// TIA Portal V17 export
// export: Created 2025-03-13T10:29:32.2184254Z, ExportSetting WithDefaults, DisplayName Totally Integrated Automation Portal, DisplayVersion V17 Update 8, DisplayName TIA Portal Openness, DisplayVersion V17 Update 8, DisplayName TIA Portal Version Control Interface, DisplayVersion V17, DisplayName SINAMICS Startdrive Advanced, DisplayVersion V17 SP2, DisplayName SINAMICS Startdrive G110M, G120, G120C, G120D, G120P, G115D, DisplayVersion V17 SP2, DisplayName SINAMICS Startdrive G130, G150, S120, S150, SINAMICS MV, S210, DisplayVersion V17 SP2, DisplayName STEP 7 Professional, DisplayVersion V17 Update 8, DisplayName SINUMERIK ONE STEP 7 Toolbox, DisplayVersion V17 Update 12, DisplayName SINUMERIK 840D sl STEP 7 Toolbox, DisplayVersion V17 Update 12, DisplayName STEP 7 Safety, DisplayVersion V17 Update 6, DisplayName WinCC Advanced, DisplayVersion V17 Update 8
FUNCTION_BLOCK "FB1801_STA3_CLEANING_VALVE"   // FB1801, LAD
{ S7_Optimized_Access := 'TRUE' }
VERSION : 0.1
// stored: AutoNumber false, IsIECCheckEnabled false, IsRetainMemResEnabled false, MemoryReserve 100, SetENOAutomatically false, UDAEnableTagReadback false
   VAR_INPUT
      SWITCH_ON_GEN_CON : Bool;
      SWITCH_ON_CON : Bool;
      SWITCH_ON_AUTO_REQ : Bool;
      SWITCH_OFF_CON : Bool;
      SWITCH_OFF_AUTO_REQ : Bool;
      HMI_LINE_REQ : Bool;
      UNIT_ALARM : UInt;
      STATION_ALARM : UInt;
   END_VAR
   VAR_OUTPUT
      SWITCHED_ON : Bool;
      SWITCHED_OFF : Bool;
      HMI_MOTION_EXECUTABILITY_LEFT : Bool;
      HMI_MOTION_EXECUTABILITY_RIGHT : Bool;
      HMI_MOTION_END_POS_LEFT : Bool;
      HMI_MOTION_END_POS_RIGHT : Bool;
      SWITCH_ON : Bool;
      SWITCH_OFF : Bool;
   END_VAR
   VAR
      VALVE : "ASPIRATION";
   END_VAR
   VAR DB_SPECIFIC
      TIMER_SIMULTANEITY { S7_SetPoint := 'True'} : TON_TIME;   // SIMULTANEITY TIMER
      TIMER_TIME_EXCEEDED { S7_SetPoint := 'True'} : TON_TIME;   // TIME EXCEEDED TIMER
   END_VAR
   VAR_TEMP
      DB_NUMBER : DInt;   // DB NUMBER FOR ALARM AND HELP DECODING
   END_VAR
   // TIMER_SIMULTANEITY.PT := T#100MS;
   // TIMER_TIME_EXCEEDED.PT := T#8S;
   VAR_TEMP   // added for the SCL form of the ladder/FBD networks
      _w1 : Bool;
      _w2 : Bool;
   END_VAR
BEGIN

REGION Network 1: GENERAL CONDITIONS
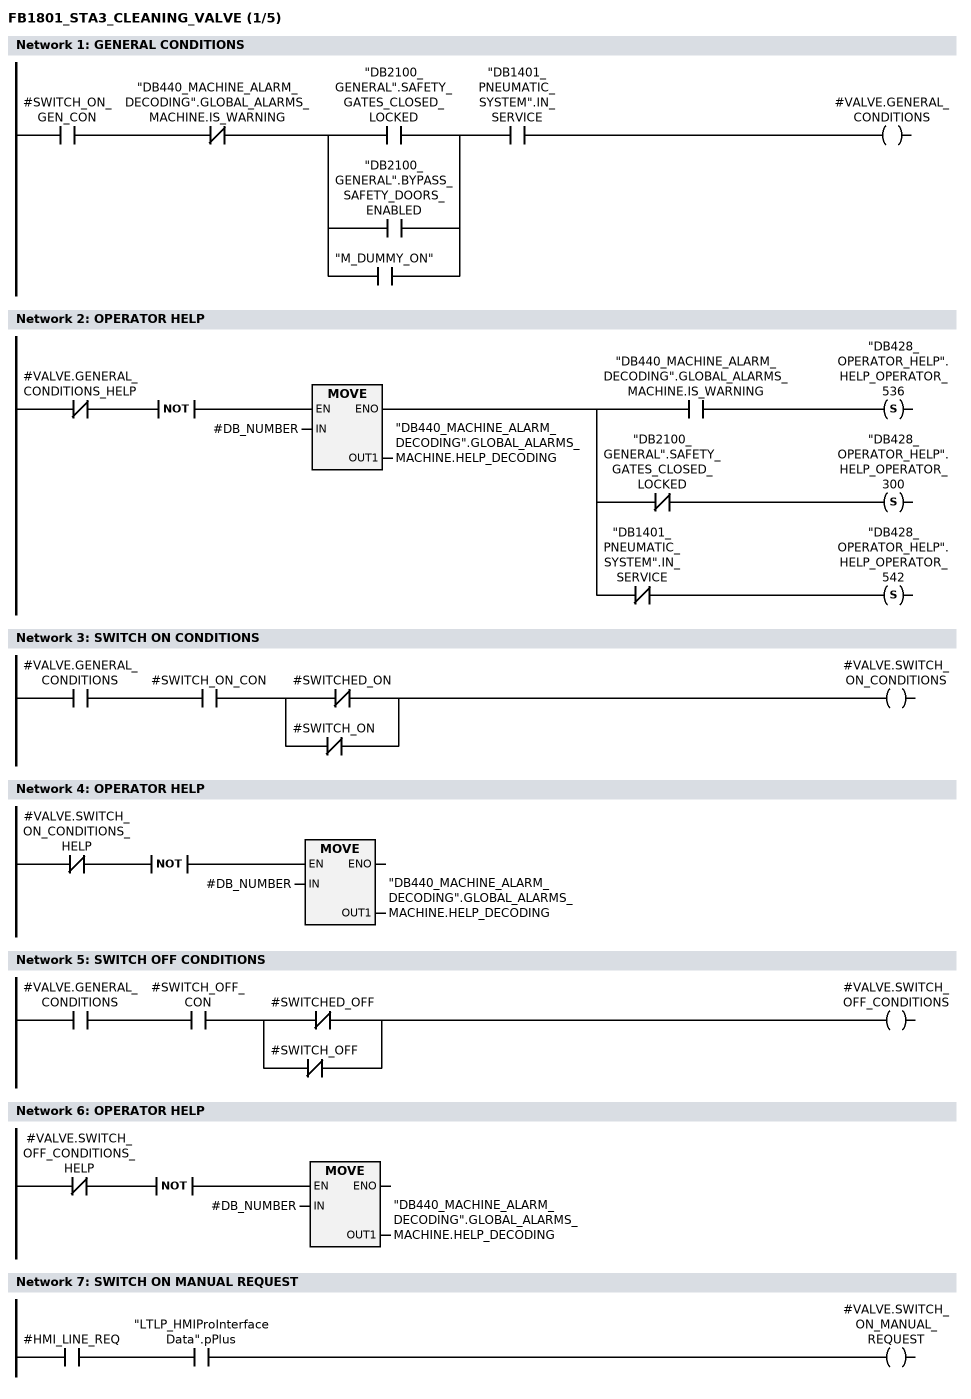
   RUNG wire#powerrail
      Contact( #SWITCH_ON_GEN_CON )
      I_Contact( "DB440_MACHINE_ALARM_DECODING".GLOBAL_ALARMS_MACHINE.IS_WARNING )
      wire#w1
      Contact( "DB2100_GENERAL".SAFETY_GATES_CLOSED_LOCKED )
      wire#w2
      Contact( "DB1401_PNEUMATIC_SYSTEM".IN_SERVICE )
      Coil( #VALVE.GENERAL_CONDITIONS )
   END_RUNG
   RUNG wire#w1
      Contact( "DB2100_GENERAL".BYPASS_SAFETY_DOORS_ENABLED )
   END_RUNG wire#w2
   RUNG wire#w1
      Contact( "M_DUMMY_ON" )
   END_RUNG wire#w2
   // the same network as SCL:
   #VALVE.GENERAL_CONDITIONS := #SWITCH_ON_GEN_CON AND NOT "DB440_MACHINE_ALARM_DECODING".GLOBAL_ALARMS_MACHINE.IS_WARNING AND ("DB2100_GENERAL".SAFETY_GATES_CLOSED_LOCKED OR "DB2100_GENERAL".BYPASS_SAFETY_DOORS_ENABLED OR "M_DUMMY_ON") AND "DB1401_PNEUMATIC_SYSTEM".IN_SERVICE;
END_REGION

REGION Network 2: OPERATOR HELP
   RUNG wire#powerrail
      I_Contact( #VALVE.GENERAL_CONDITIONS_HELP )
      Not()
      { S7_GenerateENO := "TRUE" } Move(in := #DB_NUMBER, out1 => "DB440_MACHINE_ALARM_DECODING".GLOBAL_ALARMS_MACHINE.HELP_DECODING)
      wire#w1
      Contact( "DB440_MACHINE_ALARM_DECODING".GLOBAL_ALARMS_MACHINE.IS_WARNING )
      S_Coil( "DB428_OPERATOR_HELP".HELP_OPERATOR_536 )
   END_RUNG
   RUNG wire#w1
      I_Contact( "DB2100_GENERAL".SAFETY_GATES_CLOSED_LOCKED )
      S_Coil( "DB428_OPERATOR_HELP".HELP_OPERATOR_300 )
   END_RUNG
   RUNG wire#w1
      I_Contact( "DB1401_PNEUMATIC_SYSTEM".IN_SERVICE )
      S_Coil( "DB428_OPERATOR_HELP".HELP_OPERATOR_542 )
   END_RUNG
   // the same network as SCL:
   // ENO of a box is taken as its EN; it also drops when the box reports an error
   #_w1 := NOT (NOT #VALVE.GENERAL_CONDITIONS_HELP);
   IF #_w1 THEN "DB440_MACHINE_ALARM_DECODING".GLOBAL_ALARMS_MACHINE.HELP_DECODING := #DB_NUMBER; END_IF;
   IF #_w1 AND "DB440_MACHINE_ALARM_DECODING".GLOBAL_ALARMS_MACHINE.IS_WARNING THEN
       "DB428_OPERATOR_HELP".HELP_OPERATOR_536 := TRUE;
   END_IF;
   IF #_w1 AND NOT "DB2100_GENERAL".SAFETY_GATES_CLOSED_LOCKED THEN
       "DB428_OPERATOR_HELP".HELP_OPERATOR_300 := TRUE;
   END_IF;
   IF #_w1 AND NOT "DB1401_PNEUMATIC_SYSTEM".IN_SERVICE THEN
       "DB428_OPERATOR_HELP".HELP_OPERATOR_542 := TRUE;
   END_IF;
END_REGION

REGION Network 3: SWITCH ON CONDITIONS
   RUNG wire#powerrail
      Contact( #VALVE.GENERAL_CONDITIONS )
      Contact( #SWITCH_ON_CON )
      wire#w1
      I_Contact( #SWITCHED_ON )
      wire#w2
      Coil( #VALVE.SWITCH_ON_CONDITIONS )
   END_RUNG
   RUNG wire#w1
      I_Contact( #SWITCH_ON )
   END_RUNG wire#w2
   // the same network as SCL:
   #VALVE.SWITCH_ON_CONDITIONS := #VALVE.GENERAL_CONDITIONS AND #SWITCH_ON_CON AND (NOT #SWITCHED_ON OR NOT #SWITCH_ON);
END_REGION

REGION Network 4: OPERATOR HELP
   RUNG wire#powerrail
      I_Contact( #VALVE.SWITCH_ON_CONDITIONS_HELP )
      Not()
      { S7_GenerateENO := "TRUE" } Move(in := #DB_NUMBER, out1 => "DB440_MACHINE_ALARM_DECODING".GLOBAL_ALARMS_MACHINE.HELP_DECODING)
   END_RUNG
   // the same network as SCL:
   IF NOT (NOT #VALVE.SWITCH_ON_CONDITIONS_HELP) THEN
       "DB440_MACHINE_ALARM_DECODING".GLOBAL_ALARMS_MACHINE.HELP_DECODING := #DB_NUMBER;
   END_IF;
END_REGION

REGION Network 5: SWITCH OFF CONDITIONS
   RUNG wire#powerrail
      Contact( #VALVE.GENERAL_CONDITIONS )
      Contact( #SWITCH_OFF_CON )
      wire#w1
      I_Contact( #SWITCHED_OFF )
      wire#w2
      Coil( #VALVE.SWITCH_OFF_CONDITIONS )
   END_RUNG
   RUNG wire#w1
      I_Contact( #SWITCH_OFF )
   END_RUNG wire#w2
   // the same network as SCL:
   #VALVE.SWITCH_OFF_CONDITIONS := #VALVE.GENERAL_CONDITIONS AND #SWITCH_OFF_CON AND (NOT #SWITCHED_OFF OR NOT #SWITCH_OFF);
END_REGION

REGION Network 6: OPERATOR HELP
   RUNG wire#powerrail
      I_Contact( #VALVE.SWITCH_OFF_CONDITIONS_HELP )
      Not()
      { S7_GenerateENO := "TRUE" } Move(in := #DB_NUMBER, out1 => "DB440_MACHINE_ALARM_DECODING".GLOBAL_ALARMS_MACHINE.HELP_DECODING)
   END_RUNG
   // the same network as SCL:
   IF NOT (NOT #VALVE.SWITCH_OFF_CONDITIONS_HELP) THEN
       "DB440_MACHINE_ALARM_DECODING".GLOBAL_ALARMS_MACHINE.HELP_DECODING := #DB_NUMBER;
   END_IF;
END_REGION

REGION Network 7: SWITCH ON MANUAL REQUEST
   RUNG wire#powerrail
      Contact( #HMI_LINE_REQ )
      Contact( "LTLP_HMIProInterfaceData".pPlus )
      Coil( #VALVE.SWITCH_ON_MANUAL_REQUEST )
   END_RUNG
   // the same network as SCL:
   #VALVE.SWITCH_ON_MANUAL_REQUEST := #HMI_LINE_REQ AND "LTLP_HMIProInterfaceData".pPlus;
END_REGION

REGION Network 8: SWITCH OFF MANUAL REQUEST
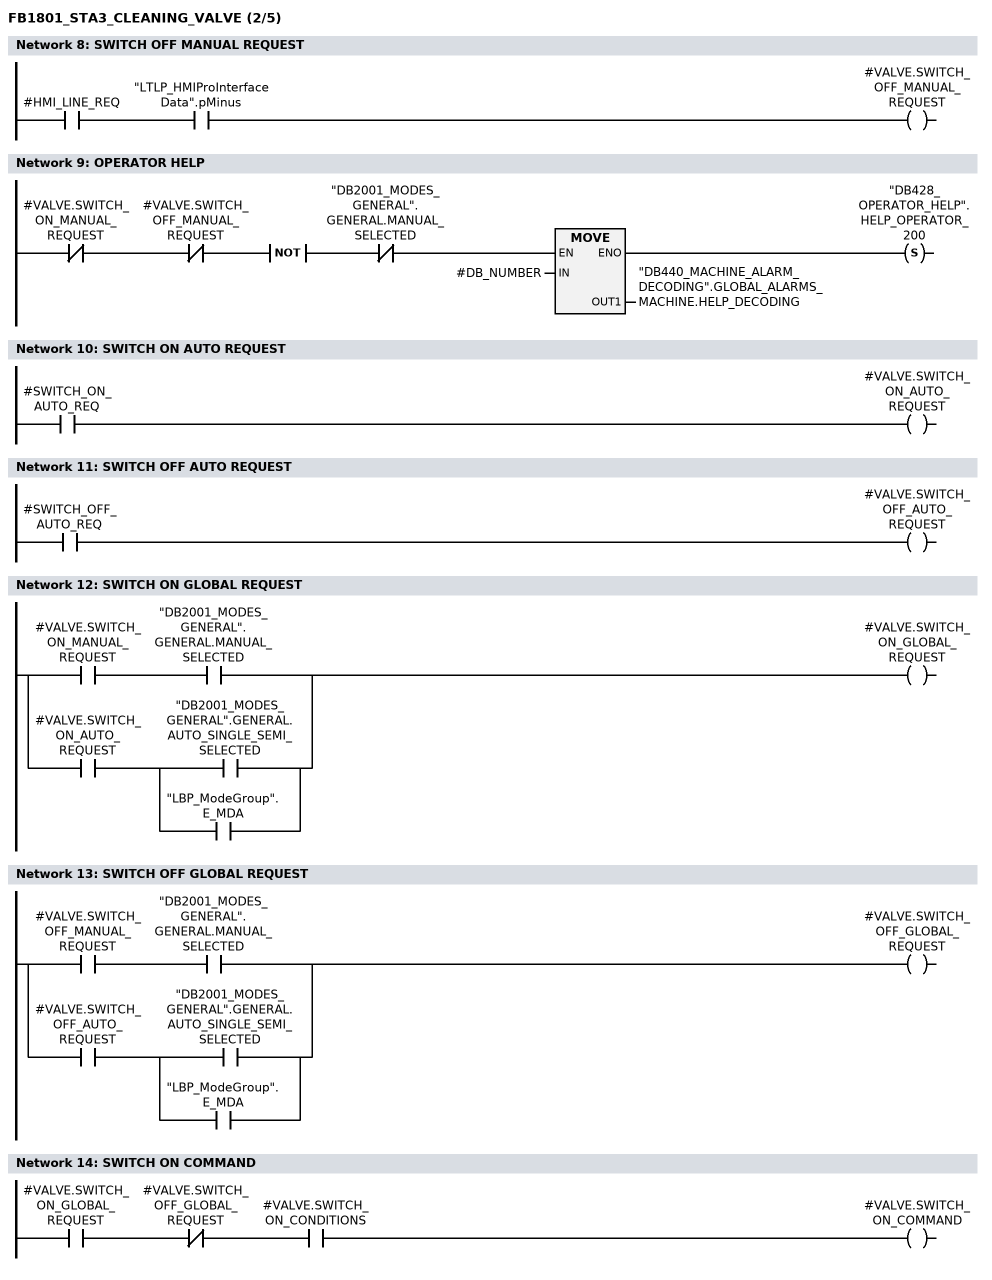
   RUNG wire#powerrail
      Contact( #HMI_LINE_REQ )
      Contact( "LTLP_HMIProInterfaceData".pMinus )
      Coil( #VALVE.SWITCH_OFF_MANUAL_REQUEST )
   END_RUNG
   // the same network as SCL:
   #VALVE.SWITCH_OFF_MANUAL_REQUEST := #HMI_LINE_REQ AND "LTLP_HMIProInterfaceData".pMinus;
END_REGION

REGION Network 9: OPERATOR HELP
   RUNG wire#powerrail
      I_Contact( #VALVE.SWITCH_ON_MANUAL_REQUEST )
      I_Contact( #VALVE.SWITCH_OFF_MANUAL_REQUEST )
      Not()
      I_Contact( "DB2001_MODES_GENERAL".GENERAL.MANUAL_SELECTED )
      { S7_GenerateENO := "TRUE" } Move(in := #DB_NUMBER, out1 => "DB440_MACHINE_ALARM_DECODING".GLOBAL_ALARMS_MACHINE.HELP_DECODING)
      S_Coil( "DB428_OPERATOR_HELP".HELP_OPERATOR_200 )
   END_RUNG
   // the same network as SCL:
   // ENO of a box is taken as its EN; it also drops when the box reports an error
   IF NOT (NOT #VALVE.SWITCH_ON_MANUAL_REQUEST AND NOT #VALVE.SWITCH_OFF_MANUAL_REQUEST) AND NOT "DB2001_MODES_GENERAL".GENERAL.MANUAL_SELECTED THEN
       "DB440_MACHINE_ALARM_DECODING".GLOBAL_ALARMS_MACHINE.HELP_DECODING := #DB_NUMBER;
       "DB428_OPERATOR_HELP".HELP_OPERATOR_200 := TRUE;
   END_IF;
END_REGION

REGION Network 10: SWITCH ON AUTO REQUEST
   RUNG wire#powerrail
      Contact( #SWITCH_ON_AUTO_REQ )
      Coil( #VALVE.SWITCH_ON_AUTO_REQUEST )
   END_RUNG
   // the same network as SCL:
   #VALVE.SWITCH_ON_AUTO_REQUEST := #SWITCH_ON_AUTO_REQ;
END_REGION

REGION Network 11: SWITCH OFF AUTO REQUEST
   RUNG wire#powerrail
      Contact( #SWITCH_OFF_AUTO_REQ )
      Coil( #VALVE.SWITCH_OFF_AUTO_REQUEST )
   END_RUNG
   // the same network as SCL:
   #VALVE.SWITCH_OFF_AUTO_REQUEST := #SWITCH_OFF_AUTO_REQ;
END_REGION

REGION Network 12: SWITCH ON GLOBAL REQUEST
   RUNG wire#powerrail
      Contact( #VALVE.SWITCH_ON_MANUAL_REQUEST )
      Contact( "DB2001_MODES_GENERAL".GENERAL.MANUAL_SELECTED )
      wire#w1
      Coil( #VALVE.SWITCH_ON_GLOBAL_REQUEST )
   END_RUNG
   RUNG wire#powerrail
      Contact( #VALVE.SWITCH_ON_AUTO_REQUEST )
      wire#w2
      Contact( "DB2001_MODES_GENERAL".GENERAL.AUTO_SINGLE_SEMI_SELECTED )
   END_RUNG wire#w1
   RUNG wire#w2
      Contact( "LBP_ModeGroup".E_MDA )
   END_RUNG wire#w1
   // the same network as SCL:
   #VALVE.SWITCH_ON_GLOBAL_REQUEST := (#VALVE.SWITCH_ON_MANUAL_REQUEST AND "DB2001_MODES_GENERAL".GENERAL.MANUAL_SELECTED) OR (#VALVE.SWITCH_ON_AUTO_REQUEST AND ("DB2001_MODES_GENERAL".GENERAL.AUTO_SINGLE_SEMI_SELECTED OR "LBP_ModeGroup".E_MDA));
END_REGION

REGION Network 13: SWITCH OFF GLOBAL REQUEST
   RUNG wire#powerrail
      Contact( #VALVE.SWITCH_OFF_MANUAL_REQUEST )
      Contact( "DB2001_MODES_GENERAL".GENERAL.MANUAL_SELECTED )
      wire#w1
      Coil( #VALVE.SWITCH_OFF_GLOBAL_REQUEST )
   END_RUNG
   RUNG wire#powerrail
      Contact( #VALVE.SWITCH_OFF_AUTO_REQUEST )
      wire#w2
      Contact( "DB2001_MODES_GENERAL".GENERAL.AUTO_SINGLE_SEMI_SELECTED )
   END_RUNG wire#w1
   RUNG wire#w2
      Contact( "LBP_ModeGroup".E_MDA )
   END_RUNG wire#w1
   // the same network as SCL:
   #VALVE.SWITCH_OFF_GLOBAL_REQUEST := (#VALVE.SWITCH_OFF_MANUAL_REQUEST AND "DB2001_MODES_GENERAL".GENERAL.MANUAL_SELECTED) OR (#VALVE.SWITCH_OFF_AUTO_REQUEST AND ("DB2001_MODES_GENERAL".GENERAL.AUTO_SINGLE_SEMI_SELECTED OR "LBP_ModeGroup".E_MDA));
END_REGION

REGION Network 14: SWITCH ON COMMAND
   RUNG wire#powerrail
      Contact( #VALVE.SWITCH_ON_GLOBAL_REQUEST )
      I_Contact( #VALVE.SWITCH_OFF_GLOBAL_REQUEST )
      Contact( #VALVE.SWITCH_ON_CONDITIONS )
      Coil( #VALVE.SWITCH_ON_COMMAND )
   END_RUNG
   // the same network as SCL:
   #VALVE.SWITCH_ON_COMMAND := #VALVE.SWITCH_ON_GLOBAL_REQUEST AND NOT #VALVE.SWITCH_OFF_GLOBAL_REQUEST AND #VALVE.SWITCH_ON_CONDITIONS;
END_REGION

REGION Network 15: SWITCH OFF COMMAND
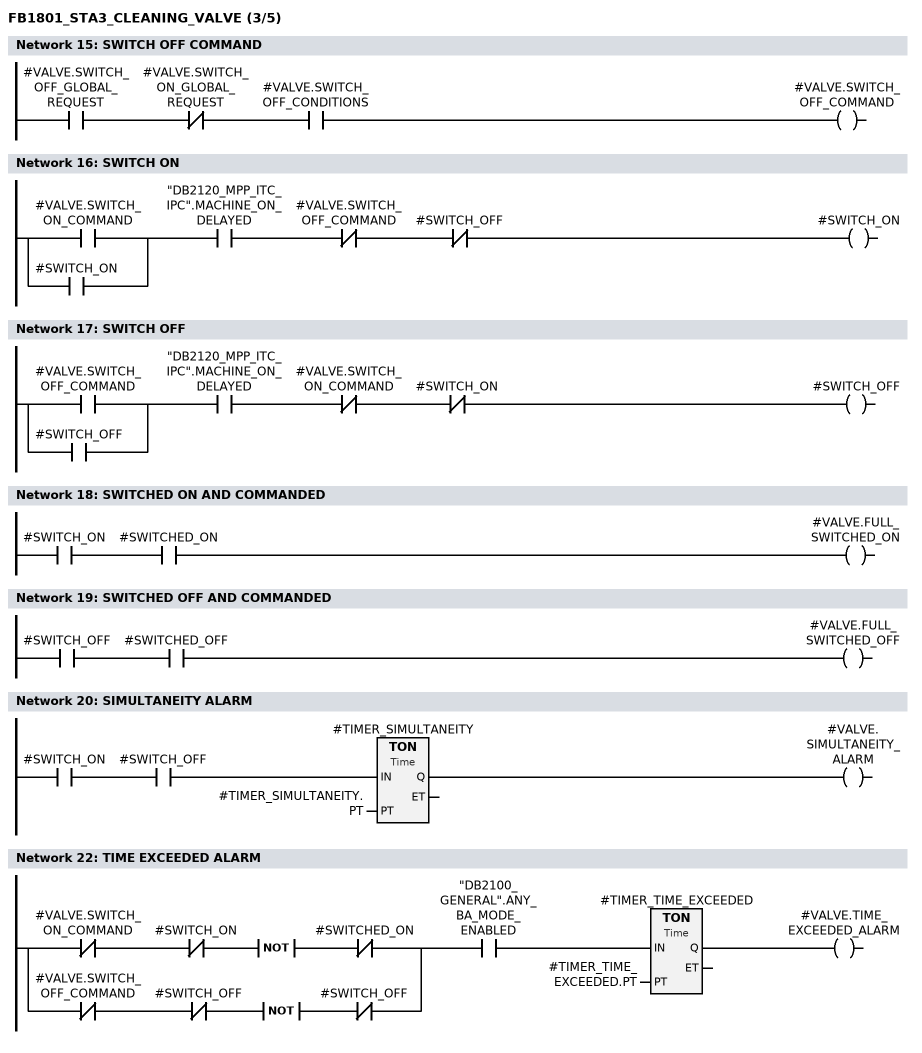
   RUNG wire#powerrail
      Contact( #VALVE.SWITCH_OFF_GLOBAL_REQUEST )
      I_Contact( #VALVE.SWITCH_ON_GLOBAL_REQUEST )
      Contact( #VALVE.SWITCH_OFF_CONDITIONS )
      Coil( #VALVE.SWITCH_OFF_COMMAND )
   END_RUNG
   // the same network as SCL:
   #VALVE.SWITCH_OFF_COMMAND := #VALVE.SWITCH_OFF_GLOBAL_REQUEST AND NOT #VALVE.SWITCH_ON_GLOBAL_REQUEST AND #VALVE.SWITCH_OFF_CONDITIONS;
END_REGION

REGION Network 16: SWITCH ON
   RUNG wire#powerrail
      Contact( #VALVE.SWITCH_ON_COMMAND )
      wire#w1
      Contact( "DB2120_MPP_ITC_IPC".MACHINE_ON_DELAYED )
      I_Contact( #VALVE.SWITCH_OFF_COMMAND )
      I_Contact( #SWITCH_OFF )
      Coil( #SWITCH_ON )
   END_RUNG
   RUNG wire#powerrail
      Contact( #SWITCH_ON )
   END_RUNG wire#w1
   // the same network as SCL:
   #SWITCH_ON := (#VALVE.SWITCH_ON_COMMAND OR #SWITCH_ON) AND "DB2120_MPP_ITC_IPC".MACHINE_ON_DELAYED AND NOT #VALVE.SWITCH_OFF_COMMAND AND NOT #SWITCH_OFF;
END_REGION

REGION Network 17: SWITCH OFF
   RUNG wire#powerrail
      Contact( #VALVE.SWITCH_OFF_COMMAND )
      wire#w1
      Contact( "DB2120_MPP_ITC_IPC".MACHINE_ON_DELAYED )
      I_Contact( #VALVE.SWITCH_ON_COMMAND )
      I_Contact( #SWITCH_ON )
      Coil( #SWITCH_OFF )
   END_RUNG
   RUNG wire#powerrail
      Contact( #SWITCH_OFF )
   END_RUNG wire#w1
   // the same network as SCL:
   #SWITCH_OFF := (#VALVE.SWITCH_OFF_COMMAND OR #SWITCH_OFF) AND "DB2120_MPP_ITC_IPC".MACHINE_ON_DELAYED AND NOT #VALVE.SWITCH_ON_COMMAND AND NOT #SWITCH_ON;
END_REGION

REGION Network 18: SWITCHED ON AND COMMANDED
   RUNG wire#powerrail
      Contact( #SWITCH_ON )
      Contact( #SWITCHED_ON )
      Coil( #VALVE.FULL_SWITCHED_ON )
   END_RUNG
   // the same network as SCL:
   #VALVE.FULL_SWITCHED_ON := #SWITCH_ON AND #SWITCHED_ON;
END_REGION

REGION Network 19: SWITCHED OFF AND COMMANDED
   RUNG wire#powerrail
      Contact( #SWITCH_OFF )
      Contact( #SWITCHED_OFF )
      Coil( #VALVE.FULL_SWITCHED_OFF )
   END_RUNG
   // the same network as SCL:
   #VALVE.FULL_SWITCHED_OFF := #SWITCH_OFF AND #SWITCHED_OFF;
END_REGION

REGION Network 20: SIMULTANEITY ALARM
   RUNG wire#powerrail
      Contact( #SWITCH_ON )
      Contact( #SWITCH_OFF )
      { S7_Templates := "time_type := Time" } #TIMER_SIMULTANEITY.TON(pt := #TIMER_SIMULTANEITY.PT, et =>)
      Coil( #VALVE.SIMULTANEITY_ALARM )
   END_RUNG
   // the same network as SCL:
   #TIMER_SIMULTANEITY(IN := #SWITCH_ON AND #SWITCH_OFF, PT := #TIMER_SIMULTANEITY.PT);   // TON
   #VALVE.SIMULTANEITY_ALARM := #TIMER_SIMULTANEITY.Q;
END_REGION

NETWORK
TITLE = READ INSTANCE DB
      L     DINO;
      +     10#800000;
      T     #DB_NUMBER;


REGION Network 22: TIME EXCEEDED ALARM
   RUNG wire#powerrail
      I_Contact( #VALVE.SWITCH_ON_COMMAND )
      I_Contact( #SWITCH_ON )
      Not()
      I_Contact( #SWITCHED_ON )
      wire#w1
      Contact( "DB2100_GENERAL".ANY_BA_MODE_ENABLED )
      { S7_Templates := "time_type := Time" } #TIMER_TIME_EXCEEDED.TON(pt := #TIMER_TIME_EXCEEDED.PT, et =>)
      Coil( #VALVE.TIME_EXCEEDED_ALARM )
   END_RUNG
   RUNG wire#powerrail
      I_Contact( #VALVE.SWITCH_OFF_COMMAND )
      I_Contact( #SWITCH_OFF )
      Not()
      I_Contact( #SWITCH_OFF )
   END_RUNG wire#w1
   // the same network as SCL:
   #TIMER_TIME_EXCEEDED(IN := ((NOT (NOT #VALVE.SWITCH_ON_COMMAND AND NOT #SWITCH_ON) AND NOT #SWITCHED_ON) OR (NOT (NOT #VALVE.SWITCH_OFF_COMMAND AND NOT #SWITCH_OFF) AND NOT #SWITCH_OFF)) AND "DB2100_GENERAL".ANY_BA_MODE_ENABLED,   // TON
                        PT := #TIMER_TIME_EXCEEDED.PT);
   #VALVE.TIME_EXCEEDED_ALARM := #TIMER_TIME_EXCEEDED.Q;
END_REGION

REGION Network 23: IMMEDIATE STOP AND STOP END OF CYCLE ALARMS
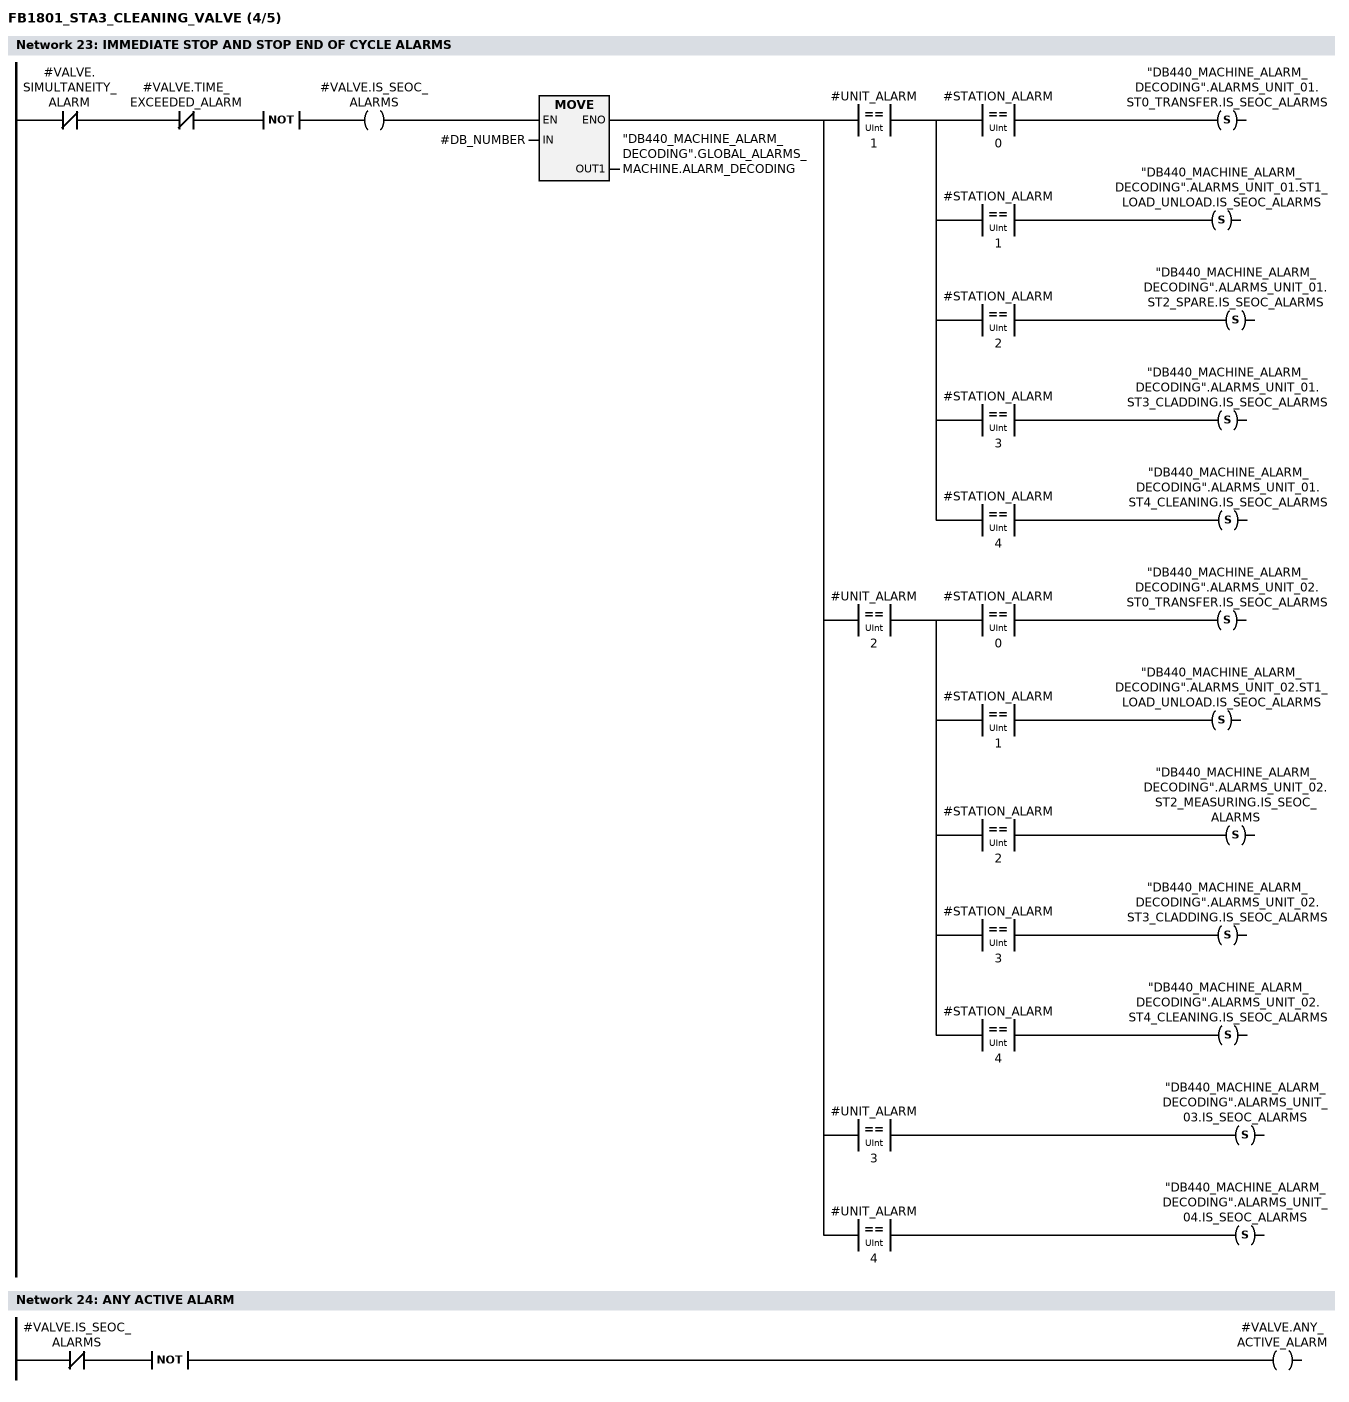
   RUNG wire#powerrail
      I_Contact( #VALVE.SIMULTANEITY_ALARM )
      I_Contact( #VALVE.TIME_EXCEEDED_ALARM )
      Not()
      Coil( #VALVE.IS_SEOC_ALARMS )
      { S7_GenerateENO := "TRUE" } Move(in := #DB_NUMBER, out1 => "DB440_MACHINE_ALARM_DECODING".GLOBAL_ALARMS_MACHINE.ALARM_DECODING)
      wire#w1
      { S7_Templates := "SrcType := UInt" } EQ_Contact(in1 := #UNIT_ALARM, in2 := 1)
      wire#w2
      { S7_Templates := "SrcType := UInt" } EQ_Contact(in1 := #STATION_ALARM, in2 := 0)
      S_Coil( "DB440_MACHINE_ALARM_DECODING".ALARMS_UNIT_01.ST0_TRANSFER.IS_SEOC_ALARMS )
   END_RUNG
   RUNG wire#w2
      { S7_Templates := "SrcType := UInt" } EQ_Contact(in1 := #STATION_ALARM, in2 := 1)
      S_Coil( "DB440_MACHINE_ALARM_DECODING".ALARMS_UNIT_01.ST1_LOAD_UNLOAD.IS_SEOC_ALARMS )
   END_RUNG
   RUNG wire#w2
      { S7_Templates := "SrcType := UInt" } EQ_Contact(in1 := #STATION_ALARM, in2 := 2)
      S_Coil( "DB440_MACHINE_ALARM_DECODING".ALARMS_UNIT_01.ST2_SPARE.IS_SEOC_ALARMS )
   END_RUNG
   RUNG wire#w2
      { S7_Templates := "SrcType := UInt" } EQ_Contact(in1 := #STATION_ALARM, in2 := 3)
      S_Coil( "DB440_MACHINE_ALARM_DECODING".ALARMS_UNIT_01.ST3_CLADDING.IS_SEOC_ALARMS )
   END_RUNG
   RUNG wire#w2
      { S7_Templates := "SrcType := UInt" } EQ_Contact(in1 := #STATION_ALARM, in2 := 4)
      S_Coil( "DB440_MACHINE_ALARM_DECODING".ALARMS_UNIT_01.ST4_CLEANING.IS_SEOC_ALARMS )
   END_RUNG
   RUNG wire#w1
      { S7_Templates := "SrcType := UInt" } EQ_Contact(in1 := #UNIT_ALARM, in2 := 2)
      wire#w3
      { S7_Templates := "SrcType := UInt" } EQ_Contact(in1 := #STATION_ALARM, in2 := 0)
      S_Coil( "DB440_MACHINE_ALARM_DECODING".ALARMS_UNIT_02.ST0_TRANSFER.IS_SEOC_ALARMS )
   END_RUNG
   RUNG wire#w3
      { S7_Templates := "SrcType := UInt" } EQ_Contact(in1 := #STATION_ALARM, in2 := 1)
      S_Coil( "DB440_MACHINE_ALARM_DECODING".ALARMS_UNIT_02.ST1_LOAD_UNLOAD.IS_SEOC_ALARMS )
   END_RUNG
   RUNG wire#w3
      { S7_Templates := "SrcType := UInt" } EQ_Contact(in1 := #STATION_ALARM, in2 := 2)
      S_Coil( "DB440_MACHINE_ALARM_DECODING".ALARMS_UNIT_02.ST2_MEASURING.IS_SEOC_ALARMS )
   END_RUNG
   RUNG wire#w3
      { S7_Templates := "SrcType := UInt" } EQ_Contact(in1 := #STATION_ALARM, in2 := 3)
      S_Coil( "DB440_MACHINE_ALARM_DECODING".ALARMS_UNIT_02.ST3_CLADDING.IS_SEOC_ALARMS )
   END_RUNG
   RUNG wire#w3
      { S7_Templates := "SrcType := UInt" } EQ_Contact(in1 := #STATION_ALARM, in2 := 4)
      S_Coil( "DB440_MACHINE_ALARM_DECODING".ALARMS_UNIT_02.ST4_CLEANING.IS_SEOC_ALARMS )
   END_RUNG
   RUNG wire#w1
      { S7_Templates := "SrcType := UInt" } EQ_Contact(in1 := #UNIT_ALARM, in2 := 3)
      S_Coil( "DB440_MACHINE_ALARM_DECODING".ALARMS_UNIT_03.IS_SEOC_ALARMS )
   END_RUNG
   RUNG wire#w1
      { S7_Templates := "SrcType := UInt" } EQ_Contact(in1 := #UNIT_ALARM, in2 := 4)
      S_Coil( "DB440_MACHINE_ALARM_DECODING".ALARMS_UNIT_04.IS_SEOC_ALARMS )
   END_RUNG
   // the same network as SCL:
   // ENO of a box is taken as its EN; it also drops when the box reports an error
   #VALVE.IS_SEOC_ALARMS := NOT (NOT #VALVE.SIMULTANEITY_ALARM AND NOT #VALVE.TIME_EXCEEDED_ALARM);
   IF #VALVE.IS_SEOC_ALARMS THEN
       "DB440_MACHINE_ALARM_DECODING".GLOBAL_ALARMS_MACHINE.ALARM_DECODING := #DB_NUMBER;
   END_IF;
   #_w1 := #VALVE.IS_SEOC_ALARMS AND (#UNIT_ALARM = 1);
   IF #_w1 AND (#STATION_ALARM = 0) THEN
       "DB440_MACHINE_ALARM_DECODING".ALARMS_UNIT_01.ST0_TRANSFER.IS_SEOC_ALARMS := TRUE;
   END_IF;
   IF #_w1 AND (#STATION_ALARM = 1) THEN
       "DB440_MACHINE_ALARM_DECODING".ALARMS_UNIT_01.ST1_LOAD_UNLOAD.IS_SEOC_ALARMS := TRUE;
   END_IF;
   IF #_w1 AND (#STATION_ALARM = 2) THEN
       "DB440_MACHINE_ALARM_DECODING".ALARMS_UNIT_01.ST2_SPARE.IS_SEOC_ALARMS := TRUE;
   END_IF;
   IF #_w1 AND (#STATION_ALARM = 3) THEN
       "DB440_MACHINE_ALARM_DECODING".ALARMS_UNIT_01.ST3_CLADDING.IS_SEOC_ALARMS := TRUE;
   END_IF;
   IF #_w1 AND (#STATION_ALARM = 4) THEN
       "DB440_MACHINE_ALARM_DECODING".ALARMS_UNIT_01.ST4_CLEANING.IS_SEOC_ALARMS := TRUE;
   END_IF;
   #_w2 := #VALVE.IS_SEOC_ALARMS AND (#UNIT_ALARM = 2);
   IF #_w2 AND (#STATION_ALARM = 0) THEN
       "DB440_MACHINE_ALARM_DECODING".ALARMS_UNIT_02.ST0_TRANSFER.IS_SEOC_ALARMS := TRUE;
   END_IF;
   IF #_w2 AND (#STATION_ALARM = 1) THEN
       "DB440_MACHINE_ALARM_DECODING".ALARMS_UNIT_02.ST1_LOAD_UNLOAD.IS_SEOC_ALARMS := TRUE;
   END_IF;
   IF #_w2 AND (#STATION_ALARM = 2) THEN
       "DB440_MACHINE_ALARM_DECODING".ALARMS_UNIT_02.ST2_MEASURING.IS_SEOC_ALARMS := TRUE;
   END_IF;
   IF #_w2 AND (#STATION_ALARM = 3) THEN
       "DB440_MACHINE_ALARM_DECODING".ALARMS_UNIT_02.ST3_CLADDING.IS_SEOC_ALARMS := TRUE;
   END_IF;
   IF #_w2 AND (#STATION_ALARM = 4) THEN
       "DB440_MACHINE_ALARM_DECODING".ALARMS_UNIT_02.ST4_CLEANING.IS_SEOC_ALARMS := TRUE;
   END_IF;
   IF #VALVE.IS_SEOC_ALARMS AND (#UNIT_ALARM = 3) THEN
       "DB440_MACHINE_ALARM_DECODING".ALARMS_UNIT_03.IS_SEOC_ALARMS := TRUE;
   END_IF;
   IF #VALVE.IS_SEOC_ALARMS AND (#UNIT_ALARM = 4) THEN
       "DB440_MACHINE_ALARM_DECODING".ALARMS_UNIT_04.IS_SEOC_ALARMS := TRUE;
   END_IF;
END_REGION

REGION Network 24: ANY ACTIVE ALARM
   RUNG wire#powerrail
      I_Contact( #VALVE.IS_SEOC_ALARMS )
      Not()
      Coil( #VALVE.ANY_ACTIVE_ALARM )
   END_RUNG
   // the same network as SCL:
   #VALVE.ANY_ACTIVE_ALARM := NOT (NOT #VALVE.IS_SEOC_ALARMS);
END_REGION

REGION Network 25: PROGRAMMING ALARM
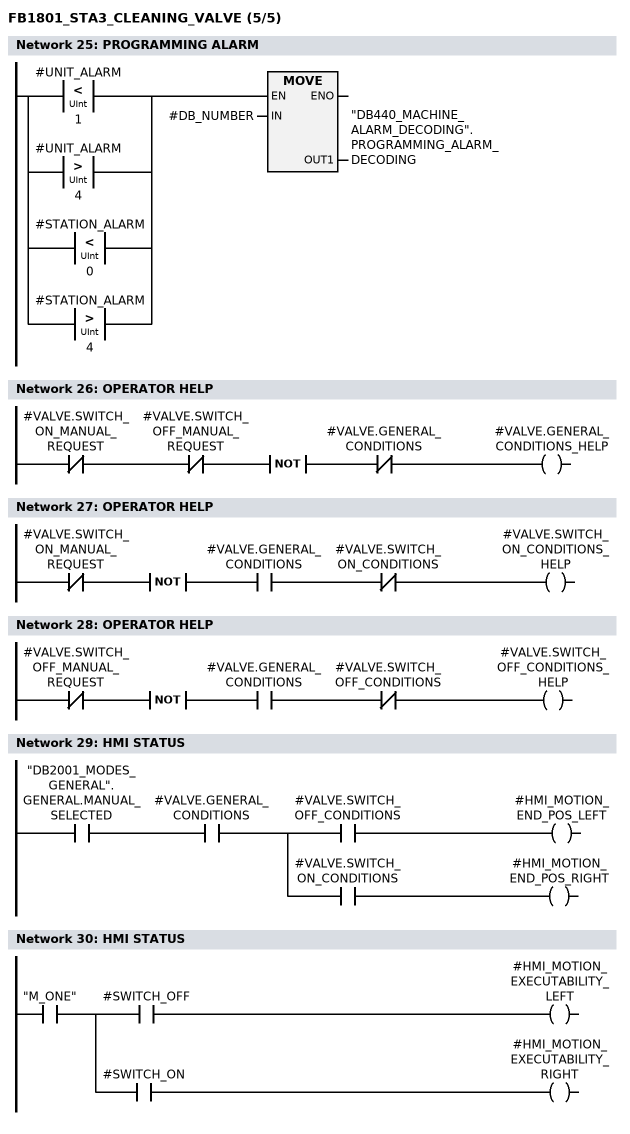
   RUNG wire#powerrail
      { S7_Templates := "SrcType := UInt" } LT_Contact(in1 := #UNIT_ALARM, in2 := 1)
      wire#w1
      Move(in := #DB_NUMBER, out1 => "DB440_MACHINE_ALARM_DECODING".PROGRAMMING_ALARM_DECODING)
   END_RUNG
   RUNG wire#powerrail
      { S7_Templates := "SrcType := UInt" } GT_Contact(in1 := #UNIT_ALARM, in2 := 4)
   END_RUNG wire#w1
   RUNG wire#powerrail
      { S7_Templates := "SrcType := UInt" } LT_Contact(in1 := #STATION_ALARM, in2 := 0)
   END_RUNG wire#w1
   RUNG wire#powerrail
      { S7_Templates := "SrcType := UInt" } GT_Contact(in1 := #STATION_ALARM, in2 := 4)
   END_RUNG wire#w1
   // the same network as SCL:
   IF (#UNIT_ALARM < 1) OR (#UNIT_ALARM > 4) OR (#STATION_ALARM < 0) OR (#STATION_ALARM > 4) THEN
       "DB440_MACHINE_ALARM_DECODING".PROGRAMMING_ALARM_DECODING := #DB_NUMBER;
   END_IF;
END_REGION

REGION Network 26: OPERATOR HELP
   RUNG wire#powerrail
      I_Contact( #VALVE.SWITCH_ON_MANUAL_REQUEST )
      I_Contact( #VALVE.SWITCH_OFF_MANUAL_REQUEST )
      Not()
      I_Contact( #VALVE.GENERAL_CONDITIONS )
      Coil( #VALVE.GENERAL_CONDITIONS_HELP )
   END_RUNG
   // the same network as SCL:
   #VALVE.GENERAL_CONDITIONS_HELP := NOT (NOT #VALVE.SWITCH_ON_MANUAL_REQUEST AND NOT #VALVE.SWITCH_OFF_MANUAL_REQUEST) AND NOT #VALVE.GENERAL_CONDITIONS;
END_REGION

REGION Network 27: OPERATOR HELP
   RUNG wire#powerrail
      I_Contact( #VALVE.SWITCH_ON_MANUAL_REQUEST )
      Not()
      Contact( #VALVE.GENERAL_CONDITIONS )
      I_Contact( #VALVE.SWITCH_ON_CONDITIONS )
      Coil( #VALVE.SWITCH_ON_CONDITIONS_HELP )
   END_RUNG
   // the same network as SCL:
   #VALVE.SWITCH_ON_CONDITIONS_HELP := NOT (NOT #VALVE.SWITCH_ON_MANUAL_REQUEST) AND #VALVE.GENERAL_CONDITIONS AND NOT #VALVE.SWITCH_ON_CONDITIONS;
END_REGION

REGION Network 28: OPERATOR HELP
   RUNG wire#powerrail
      I_Contact( #VALVE.SWITCH_OFF_MANUAL_REQUEST )
      Not()
      Contact( #VALVE.GENERAL_CONDITIONS )
      I_Contact( #VALVE.SWITCH_OFF_CONDITIONS )
      Coil( #VALVE.SWITCH_OFF_CONDITIONS_HELP )
   END_RUNG
   // the same network as SCL:
   #VALVE.SWITCH_OFF_CONDITIONS_HELP := NOT (NOT #VALVE.SWITCH_OFF_MANUAL_REQUEST) AND #VALVE.GENERAL_CONDITIONS AND NOT #VALVE.SWITCH_OFF_CONDITIONS;
END_REGION

REGION Network 29: HMI STATUS
   RUNG wire#powerrail
      Contact( "DB2001_MODES_GENERAL".GENERAL.MANUAL_SELECTED )
      Contact( #VALVE.GENERAL_CONDITIONS )
      wire#w1
      Contact( #VALVE.SWITCH_OFF_CONDITIONS )
      Coil( #HMI_MOTION_END_POS_LEFT )
   END_RUNG
   RUNG wire#w1
      Contact( #VALVE.SWITCH_ON_CONDITIONS )
      Coil( #HMI_MOTION_END_POS_RIGHT )
   END_RUNG
   // the same network as SCL:
   #_w1 := "DB2001_MODES_GENERAL".GENERAL.MANUAL_SELECTED AND #VALVE.GENERAL_CONDITIONS;
   #HMI_MOTION_END_POS_LEFT := #_w1 AND #VALVE.SWITCH_OFF_CONDITIONS;
   #HMI_MOTION_END_POS_RIGHT := #_w1 AND #VALVE.SWITCH_ON_CONDITIONS;
END_REGION

REGION Network 30: HMI STATUS
   RUNG wire#powerrail
      Contact( "M_ONE" )
      wire#w1
      Contact( #SWITCH_OFF )
      Coil( #HMI_MOTION_EXECUTABILITY_LEFT )
   END_RUNG
   RUNG wire#w1
      Contact( #SWITCH_ON )
      Coil( #HMI_MOTION_EXECUTABILITY_RIGHT )
   END_RUNG
   // the same network as SCL:
   #HMI_MOTION_EXECUTABILITY_LEFT := "M_ONE" AND #SWITCH_OFF;
   #HMI_MOTION_EXECUTABILITY_RIGHT := "M_ONE" AND #SWITCH_ON;
END_REGION
END_FUNCTION_BLOCK
